# EPICS StreamDevice protocol: EPICS/Db/aim.proto
# Author: Philip Weigel

Terminator = CR;

get_pressure {
	out "?V752";
	in "=V752 %e;%*d";
}

enable {
	out "!C752";
	in "!%d";
}
